FUNCTION_BLOCK MOTOR_F_B (* Service Interface Function Block Type *)
  (* Standard: 61499-2 *)
  (* Version 1.0, 2019-04-05, adeel *)
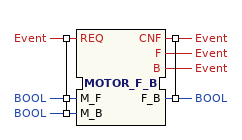
  EVENT_INPUT
    REQ WITH M_F, M_B; (* Service Request *)
  END_EVENT
  EVENT_OUTPUT
    CNF WITH F_B; (* Confirmation of Requested Service *)
    F; (* FORWARD *)
    B; (* BACKWARD *)
  END_EVENT
  VAR_INPUT
    M_F : BOOL; (* MOVE FORWARD *)
    M_B : BOOL;
  END_VAR
  VAR_OUTPUT
    F_B : BOOL;
  END_VAR
  SERVICE APPLICATION/RESOURCE (* Service Interface Function Block Type *)
    SEQUENCE normal_establishment
      APPLICATION.INIT+(PARAMS) -> RESOURCE.initialize(PARAMS) -> APPLICATION.INITO+();
    END_SEQUENCE
    SEQUENCE unsuccessful_establishment
      APPLICATION.INIT+(PARAMS) -> RESOURCE.initialize(PARAMS) -> APPLICATION.INITO-(STATUS);
    END_SEQUENCE
    SEQUENCE request_confirm
      APPLICATION.REQ+(SD) -> RESOURCE.request(SD) -> APPLICATION.CNF+(RD);
    END_SEQUENCE
    SEQUENCE request_inhibited
      APPLICATION.REQ-(SD) -> APPLICATION.CNF-(STATUS);
    END_SEQUENCE
    SEQUENCE request_error
      APPLICATION.REQ+(SD) -> RESOURCE.request(SD) -> APPLICATION.CNF-(STATUS);
    END_SEQUENCE
    SEQUENCE indication_response
      RESOURCE.indicate(RD) -> APPLICATION.IND+(RD);
      APPLICATION.RSP(QI,SD) -> RESOURCE.response(QI,SD);
    END_SEQUENCE
    SEQUENCE indication_inhibited
      RESOURCE.indicate(RD,QI=FALSE) -> RESOURCE.inhibited();
    END_SEQUENCE
    SEQUENCE error_indication
      RESOURCE.error(STATUS) -> APPLICATION.IND-(STATUS);
    END_SEQUENCE
    SEQUENCE application_initiated_termination
      APPLICATION.INIT-() -> RESOURCE.terminate() -> APPLICATION.INITO-(STATUS);
    END_SEQUENCE
    SEQUENCE resource_initiated_termination
      -> APPLICATION.INITO-(STATUS);
    END_SEQUENCE
  END_SERVICE
END_FUNCTION_BLOCK
